PROGRAM AxisVertical
VAR_INPUT
	Desired_Speed: INT ;
	Desired_Position: UINT ;
	tolerance: UINT;
END_VAR
VAR
	Axis : ST_Axis := (
		uiCounterValue := INPUT.IW_VGR_CounterValueVertical,
		bSetCounter := OUTPUT.QX_VGR_SetCounterVertical,
		uiSetCounterValue := OUTPUT.QW_VGR_SetCounterValueVertical,
		iControl := VGR.QW_VGR_PWM_Vertical_Control,
		iPWM := VGR.QW_VGR_PWM_Vertical_M1,
		bJogMinus := VGR.QX_VGR_M1_VerticalAxisUp_Q1,
		bJogPlus := VGR.QX_VGR_M1_VerticalAxisDown_Q2
	);
	
	Motor_Direction_Vertical: Motor_direction;
END_VAR

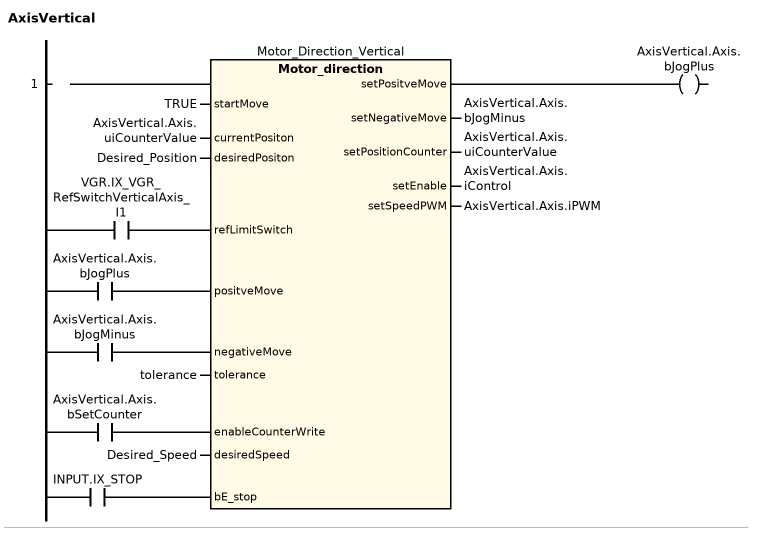
// NETWORK 1
Motor_Direction_Vertical(
    startMove := TRUE,
    currentPositon := AxisVertical.Axis.uiCounterValue,
    desiredPositon := Desired_Position,
    refLimitSwitch := VGR.IX_VGR_RefSwitchVerticalAxis_I1,
    positveMove := AxisVertical.Axis.bJogPlus,
    negativeMove := AxisVertical.Axis.bJogMinus,
    tolerance := tolerance,
    enableCounterWrite := AxisVertical.Axis.bSetCounter,
    desiredSpeed := Desired_Speed,
    bE_stop := INPUT.IX_STOP,
    setNegativeMove => AxisVertical.Axis.bJogMinus,
    setPositionCounter => AxisVertical.Axis.uiCounterValue,
    setEnable => AxisVertical.Axis.iControl,
    setSpeedPWM => AxisVertical.Axis.iPWM); // Motor_direction
AxisVertical.Axis.bJogPlus := Motor_Direction_Vertical.setPositveMove;

END_PROGRAM

(* stored: Version 1.1.0.1, ProductVersion 3.1.4024.12
   POU AxisVertical: Id {d3a4e310-1599-411c-abd2-dad3586ecff7}, SpecialFunc None *)
